FUNCTION_BLOCK PB_NOpen IMPLEMENTS I_PB
VAR
	bInput AT %I* :BOOL;
	
END_VAR

PROPERTY IsPressed : BOOL
//Property of PB when pressed
GET
VAR
	//Giving the properties of bInputSensor to isPressed
END_VAR
IsPressed := bInput;
END_GET
END_PROPERTY

PROPERTY IsReleased : BOOL
//Property of PB when PBNOpen is released
GET
VAR
	//Giving the properties of bInputSensor to isPressed
END_VAR
IsReleased := NOT bInput;
END_GET
END_PROPERTY

END_FUNCTION_BLOCK

(* stored: Version 1.1.0.1, ProductVersion 3.1.4024.12
   POU PB_NOpen: Id {44309809-c3cd-43c2-937b-a5a2e61b4600}, SpecialFunc None
   Property IsPressed: Id {436d6bab-f1cc-467b-a463-c09895f1697e}
   Get Get: Id {04f67856-0578-4e63-b66b-94192e1d7d22}
   Property IsReleased: Id {6f3903d3-47b5-4b37-a1b4-9acd7eb2f282}
   Get Get: Id {7c03c24d-fde5-402c-a6ba-0b77a6d5f407} *)
